{attribute addProperty BoxType "EL6851-0000-0017"}
{attribute addProperty Id "Transmit_requestAT %Q*BOOL811Disable_cyclic_TxDAT %Q*BOOL813Send_default_dataAT %Q*BOOL814Channel_lengthAT %Q*UINT16217Start_codeAT %Q*USINT8118"}
{attribute addProperty CRC "1808455154"}
{attribute addProperty SizeInBites "48"}
{attribute addProperty SizeInBytes "6"}
TYPE DMX_Control_6BCAD5F2 :
STRUCT
	{attribute addProperty Name "Transmit_request"}
	Transmit_request AT %Q* : BOOL;
	{attribute addProperty Name "Disable_cyclic_TxD"}
	Disable_cyclic_TxD AT %Q* : BOOL;
	{attribute addProperty Name "Send_default_data"}
	Send_default_data AT %Q* : BOOL;
	{attribute addProperty Name "Channel_length"}
	Channel_length AT %Q* : UINT;
	{attribute addProperty Name "Start_code"}
	Start_code AT %Q* : USINT;
END_STRUCT
END_TYPE

(* stored: Version 1.2.0.0, ProductVersion 3.1.4024.9
   DUT DMX_Control_6BCAD5F2: Id {5607e790-8f40-4659-a5e6-55f9421e0acd} *)
